INTERFACE I_Filter

METHOD SetFilter : BOOL
VAR_INPUT
	FilterPos	: USINT;
END_VAR
END_METHOD

END_INTERFACE

(* stored: Version 1.1.0.1, ProductVersion 3.1.4024.12
   Itf I_Filter: Id {7e4f80b1-b6cc-4387-86b4-3956422cdca3}
   Method SetFilter: Id {6999e10a-d22d-4416-aea3-af5c082017db} *)
